FUNCTION_BLOCK CTRL_PI (* FT_PI is a PI controller with manual functionality. *)
  (* Standard: 61499-2; Description: version 2.0	30. jun 2008 programmer 	hugo tested by	oscat FT_PI is a PI controller with manual functionality. The PID controller works according to the fomula Y = e *(KP+ KI * INTEG(e) ) + offset, while e = set_point - actual. a rst will reset all internal data, while a switch to manual will cause the controller to follow the function Y = manual_in + offset. limit_h and Limit_l set the possible output range of Y. the output flags lim will signal that the output limits are active and overflow will signal that the integrator has reached its limits. since rev 1.1 the "trapezregel is used for more accuracy. rev 1.2 added selective integratin which means the integrative component is only active within a small range of the target value this avoids the integrator to go to limits while an input setpoint change happened and is only causing overshoots. the int_band is by default 100 which means the int is active all the time and if set to for example to 0.1 the integrator is only active while the input is between 0.9 and 1.1 of the set_point value. default values for KP = 1, TN = 1, TV = 1, LIMIT_L = -1000, LIMIT_H = +1000. *)
  (* Version 1.0, 2025-12-19, franz *)
  PACKAGE OSCAT::Basic::POUs::Engineering::Control;
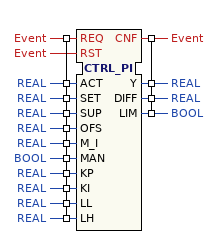
  EVENT_INPUT
    REQ WITH ACT, SET, SUP, OFS, M_I, MAN, KP, KI, LL, LH; (* Normal Execution Request *)
    RST; (* Reset *)
  END_EVENT
  EVENT_OUTPUT
    CNF WITH Y, DIFF, LIM; (* Execution Confirmation *)
  END_EVENT
  VAR_INPUT
    ACT : REAL; (* Actual Value *)
    SET : REAL; (* Set Point *)
    SUP : REAL; (* Noise Suppression *)
    OFS : REAL; (* Offset *)
    M_I : REAL; (* Manual Input Value *)
    MAN : BOOL; (* Manual Mode *)
    KP : REAL := 1.0; (* Proportional Gain *)
    KI : REAL := 1.0; (* Integral Gain *)
    LL : REAL := -1000.0; (* Lower Limit *)
    LH : REAL := 1000.0; (* Upper Limit *)
  END_VAR
  VAR_OUTPUT
    Y : REAL; (* Control Output *)
    DIFF : REAL; (* Difference (Error) *)
    LIM : BOOL; (* Limit Reached Flag *)
  END_VAR
  FBS
    pi : OSCAT::Basic::POUs::Engineering::Control::FT_PIWL; (* Internal PI controller *)
    co : OSCAT::Basic::POUs::Engineering::Control::CTRL_OUT; (* Internal Control Output Instance *)
  END_FBS
  EC_STATES
    REQ : REQ -> CNF;
    RST : RST -> CNF;
  END_STATES
  ALGORITHM RST IN ST:
pi.RST();
  END_ALGORITHM
  ALGORITHM REQ IN ST:
ALGORITHM REQ
DIFF := CTRL_IN(SET, ACT, SUP);
pi.REQ(in := DIFF, kp := KP, ki := KI, lim_l := LL, lim_h := LH);
co(ci := pi.Y, OFFSET := OFS, man_in := M_I, lim_l := LL, lim_h := LH, MANUAL := MAN);
Y := co.Y;
LIM := co.LIM;
END_ALGORITHM

(* revision history hm 	31.10.2007 		rev 1.0 original version
 * *
 * hm	3.11.2007		rev 1.1 added noise input to filter noise added output diff set limit output
 * false when output is within limits overfolw was not set correctly
 * *
 * hm	5. jan 2008		rev 1.2 improved performance
 * *
 * hm	20. jun. 2008	rev 2.0 rewritten using new modular approach *)
  END_ALGORITHM
END_FUNCTION_BLOCK
